VAR_GLOBAL
    {attribute 'pytmc' := '
        pv: PLC:KFE:RIX:VAC:K2:FFO:02
    '}
    {attribute 'TcLinkTo' := '.q_xFastFaultOut:=TIIB[PMPS_FFO (EL2202)]^Channel 2^Output'}
    g_FastFaultOutput2  :	FB_HardwareFFOutput:= (i_sNetID:='172.21.42.126.1.1');	//FFO for Fast Shutter Valves upstream of ST1K2_PPS
END_VAR

(* stored: Version 1.1.0.1, ProductVersion 3.1.4022.18
   GVL GVL_RIX_VAC_FSV_PMPS: Id {ed2ee3c9-b45b-4b97-b27e-aec2da38456b} *)
